// TwinCAT 3 PLC project MCAG_PLC_Project
// ProgramVersion: 3.1.0.8
// libraries:
//   Tc2_MC2, * (Beckhoff Automation GmbH)
//   Tc2_Standard, * (Beckhoff Automation GmbH)
//   Tc2_System, * (Beckhoff Automation GmbH)
//   Tc2_Utilities, * (Beckhoff Automation GmbH)
//   Tc3_Interfaces, * (Beckhoff Automation GmbH)
//   Tc3_Module, * (Beckhoff Automation GmbH)
// project tree:
//   DUTs/ DUT_AxisStatus_v0_01.TcDUT (not stored), DUT_AxisStatus_v0_02.TcDUT (not stored)
//   / PlcTask.TcTTO (not stored)
//   POUs/ FB_ReadFloatParameter.TcPOU (not stored), FB_ReadParameterInNc_v1_00.TcPOU (not stored), FB_WriteParameterInNc_v1_00.TcPOU (not stored), MAIN.TcPOU
//   POUs/Hardware/EtherCAT_Terminals/Analog_Inputs/ FB_CalculateFrequency_3702_v0_01.TcPOU (not stored), FB_EL3702_v0_00.TcPOU (not stored), FB_EL3773_v0_00.TcPOU (not stored), FB_EL3773_v1_00.TcPOU (not stored)
//   POUs/Hardware/EtherCAT_Terminals/Digital_Inputs/ EL1002_v1_00.TcPOU (not stored), EL1004_v1_00.TcPOU (not stored), EL1008_v1_00.TcPOU (not stored), EL1012_v1_00.TcPOU (not stored), EL1014_v1_00.TcPOU (not stored), EL1018_v1_00.TcPOU (not stored), EL1024_v1_00.TcPOU (not stored), EL1034_v1_00.TcPOU (not stored), EL1084_v1_00.TcPOU (not stored), EL1088_v1_00.TcPOU (not stored), EL1094_v1_00.TcPOU (not stored), EL1098_v1_00.TcPOU (not stored), EL1104_v1_00.TcPOU (not stored), EL1114_v1_00.TcPOU (not stored), EL1124_v1_00.TcPOU (not stored), EL1134_v1_00.TcPOU (not stored), EL1144_v1_00.TcPOU (not stored), EL1202_v1_00.TcPOU (not stored), EL1252_v1_00.TcPOU (not stored), EL1258_v0_00.TcPOU (not stored), EL1259_v0_00.TcPOU (not stored), EL1262_v0_00.TcPOU (not stored), EL1502_v0_00.TcPOU (not stored), EL1512_v0_00.TcPOU (not stored), EL1702_v1_00.TcPOU (not stored), EL1712_v1_00.TcPOU (not stored), EL1722_v1_00.TcPOU (not stored), EL1804_v1_00.TcPOU (not stored), EL1808_v1_00.TcPOU (not stored), EL1809_v1_00.TcPOU (not stored), EL1814_v1_00.TcPOU (not stored), EL1819_v1_00.TcPOU (not stored), EL1859_v1_00.TcPOU (not stored), EL1862_v1_00.TcPOU (not stored), EL1872_v1_00.TcPOU (not stored), EL1889_v1_00.TcPOU (not stored), FB_EL1008_v1_00.TcPOU (not stored), FB_EL1202_v1_00.TcPOU (not stored), FB_EL1252ASM_v1_00.TcPOU (not stored), FB_EL1252_v1_00.TcPOU (not stored)
//   POUs/Hardware/EtherCAT_Terminals/Digital_Outputs/ EL2002_v1_00.TcPOU (not stored), EL2004_v1_00.TcPOU (not stored), EL2008_v1_00.TcPOU (not stored), EL2022_v1_00.TcPOU (not stored), EL2024_v1_00.TcPOU (not stored), EL2032_v1_00.TcPOU (not stored), EL2034_v1_00.TcPOU (not stored), EL2042_v1_00.TcPOU (not stored), EL2084_v1_00.TcPOU (not stored), EL2088_v1_00.TcPOU (not stored), EL2124_v1_00.TcPOU (not stored), EL2202_v0_00.TcPOU (not stored), EL2212_v0_00.TcPOU (not stored), EL2252_v0_00.TcPOU (not stored), EL2258_v0_00.TcPOU (not stored), EL2262_v0_00.TcPOU (not stored), EL2502_v0_00.TcPOU (not stored), EL2521_v1_00.TcPOU (not stored), EL2535_v0_00.TcPOU (not stored), FB_EL2008_v1_00.TcPOU (not stored)
//   POUs/Hardware/EtherCAT_Terminals/Digital_Outputs/External_Types/ dutEL2521_Ctrl.TcDUT (not stored), dutEL2521_Status.TcDUT (not stored)
//   POUs/Hardware/EtherCAT_Terminals/Digital_Outputs/Safety_Terminals/ EL1904_v0_00.TcPOU (not stored), EL1908_v0_00.TcPOU (not stored), EL2901_v0_00.TcPOU (not stored), EL2902_v0_00.TcPOU (not stored), EL2904_v0_00.TcPOU (not stored), EL2964_v0_00.TcPOU (not stored), EL6900_v0_00.TcPOU (not stored), FB_EL1904_v1_00.TcPOU (not stored), FB_EL2904_v1_00.TcPOU (not stored), FB_EL6900_v1_00.TcPOU (not stored)
//   POUs/Hardware/EtherCAT_Terminals/Motion/ EL7211_v1_00.TcPOU (not stored), EL9576_v1_00.TcPOU (not stored)
//   POUs/Hardware/EtherCAT_Terminals/System/ EL9505_V1_00.TcPOU (not stored)
//   POUs/Hardware/Other/ EK1200.TcPOU (not stored)
//   POUs/Motion/ FB_DriveVirtual.TcPOU (not stored), FB_NcAxis.TcPOU (not stored)
// real-time tasks:
//   TASK PlcTask: cycle T#10ms, priority 20, ADS port 350
//   TASK PlcTaskCom: cycle T#1ms, priority 26, ADS port 351
// motion (NC):
//   TASK NC-Task 1 SAF: cycle T#2ms, priority 4, ADS port 501
//   TASK NC-Task 1 SVB: cycle T#10ms, priority 8, ADS port 511
//   AXIS Axis 1 (id 1)
//     Velo: RefSearch=10, RefSync=5
//     PositionAreaControl: Enable=false, RefSearch=false
//     OtherSettings: AllowMotionCmdToSlave=true
//     encoder EncType=8
//       EncPara: ScaleFactorNumerator=60, ScaleFactorDenominator=12800, MaxCount=#xffffffff
//     encoder EncId=129, EncType=4
//       EncPara: ScaleFactorNumerator=70, ScaleFactorDenominator=4096, Inverse=true, MaxCount=#x0000ffff
//         Inc: RefMode=2, RefSoftSyncMask=#x0000ffff
//     drive DrvType=9
//       DrvPara: MaxCount=#xffffffff, DriveControlDWord=#x00030100
//         Analog: VeloScale=1.02400649589962
//         TimeComp: TaskDelayCycles=1
//     controller CtrType=1
//       CtrPara: PriorControlFactor=1
//         PosDiffControl: Enable=false
//         PID: PosKp=10
//         Observer: BandWidth=20
//   AXIS Axis 2 (id 2)
//     OtherSettings: AllowMotionCmdToSlave=true
//     encoder EncType=8
//       EncPara: MaxCount=#x0036ee7f
//     drive DrvType=9
//       DrvPara: MaxCount=#xffffffff
//         Analog: VeloScale=6
//         TimeComp: TaskDelayCycles=1
//     controller CtrType=1
//       CtrPara: PriorControlFactor=1
//         Observer: BandWidth=20
//   AXIS Axis 3 (id 3)
//     OtherSettings: AllowMotionCmdToSlave=true
//     encoder EncType=1
//     drive DrvType=5
//       TimeComp: TaskDelayCycles=1
//     controller CtrType=1
//       CtrPara: PriorControlFactor=1
//         Observer: BandWidth=20
//   AXIS Axis 4 (id 4)
//     OtherSettings: AllowMotionCmdToSlave=true
//     encoder EncType=8
//       EncPara: MaxCount=#xffffffff
//     drive DrvType=9
//       DrvPara: MaxCount=#xffffffff, DriveControlDWord=#x00030100
//         Analog: VeloScale=1.02400649589962
//         TimeComp: TaskDelayCycles=1
//     controller CtrType=1
//       CtrPara: PriorControlFactor=1
//         Observer: BandWidth=20
// I/O:
//   DEVICE Device 1 (EtherCAT), AmsNetId 5.29.123.218.2.1
//     Term 1 (EK1200) [EK1200-5000 EtherCAT Power supply (2A E-Bus)]
//       Term 2 (EK1110) [EK1110 EtherCAT extension]
//     Drive 3 (AX5021-0000-0001) [AX5021-0000 EtherCAT Drive (SoE, 1 Ch.)]
//     Drive 4 (AX5112-0000-0203) [AX5112-0000-0203 EtherCAT Drive (SoE, 1 Ch.)]
//     Drive 5 (AX5112-0000-0203) [AX5112-0000-0203 EtherCAT Drive (SoE, 1 Ch.)]
// variable links:
//   NC-Task 1 SAF/Axes/Axis 1 <-> Device 1 (EtherCAT)/Drive 4 (AX5112-0000-0203)
//     Drive/Inputs/In/nDataIn1 <-> AT/Following distance
//     Drive/Inputs/In/nDcOutputTime <-> InfoData/DcOutputShift
//     Drive/Inputs/In/nState1 <-> AT/Drive status word @bit 8
//     Drive/Inputs/In/nState2 <-> AT/Drive status word
//     Drive/Inputs/In/nState4 @bit 1 <-> WcState/InputToggle
//     Drive/Inputs/In/nState4 <-> WcState/WcState
//     Drive/Outputs/Out/nCtrl1 <-> MDT/Master control word @bit 8
//     Drive/Outputs/Out/nDataOut1 <-> MDT/Position command value
//     Enc/Inputs/In/nDataIn1 <-> AT/Position feedback 1 value
//     Enc/Inputs/In/nDcInputTime <-> InfoData/DcInputShift
//     Enc/Inputs/In/nState4 @bit 1 <-> WcState/InputToggle
//     Enc/Inputs/In/nState4 <-> WcState/WcState
//   NC-Task 1 SAF/Axes/Axis 2 <-> Device 1 (EtherCAT)/Drive 3 (AX5021-0000-0001)
//     Drive/Inputs/In/nDcOutputTime <-> InfoData/DcOutputShift
//     Drive/Inputs/In/nState1 <-> AT/Drive status word @bit 8
//     Drive/Inputs/In/nState2 <-> AT/Drive status word
//     Drive/Inputs/In/nState4 @bit 1 <-> WcState/InputToggle
//     Drive/Inputs/In/nState4 <-> WcState/WcState
//     Drive/Outputs/Out/nCtrl1 <-> MDT/Master control word @bit 8
//     Enc/Inputs/In/nDcInputTime <-> InfoData/DcInputShift
//     Enc/Inputs/In/nState4 @bit 1 <-> WcState/InputToggle
//     Enc/Inputs/In/nState4 <-> WcState/WcState
//   NC-Task 1 SAF/Axes/Axis 4 <-> Device 1 (EtherCAT)/Drive 5 (AX5112-0000-0203)
//     Drive/Inputs/In/nDataIn1 <-> AT/Following distance
//     Drive/Inputs/In/nDcOutputTime <-> InfoData/DcOutputShift
//     Drive/Inputs/In/nState1 <-> AT/Drive status word @bit 8
//     Drive/Inputs/In/nState2 <-> AT/Drive status word
//     Drive/Inputs/In/nState4 @bit 1 <-> WcState/InputToggle
//     Drive/Inputs/In/nState4 <-> WcState/WcState
//     Drive/Outputs/Out/nCtrl1 <-> MDT/Master control word @bit 8
//     Drive/Outputs/Out/nDataOut1 <-> MDT/Position command value
//     Enc/Inputs/In/nDataIn1 <-> AT/Position feedback 1 value
//     Enc/Inputs/In/nDcInputTime <-> InfoData/DcInputShift
//     Enc/Inputs/In/nState4 @bit 1 <-> WcState/InputToggle
//     Enc/Inputs/In/nState4 <-> WcState/WcState
//   MCAG_PLC_Project/MCAG_PLC_Project Instance <-> NC-Task 1 SAF/Axes/Axis 1
//     PlcTask Inputs/MAIN.M1Link.Axis.NcToPlc <-> Outputs/ToPlc
//     PlcTask Outputs/MAIN.M1Link.Axis.PlcToNc <-> Inputs/FromPlc

// ---- POUs/MAIN.TcPOU
PROGRAM MAIN
VAR
	sVersion: STRING:='1.0.0';
	M1:FB_DriveVirtual;
	M1Link:FB_NcAxis;
	M2:FB_DriveVirtual;
	M2Link:FB_NcAxis;
	bLimitFwd AT %I*: BOOL;
	bLimitBwd AT %I*: BOOL;
	bHomeSensor AT %I*: BOOL;
END_VAR

act();

ACTION ACT:
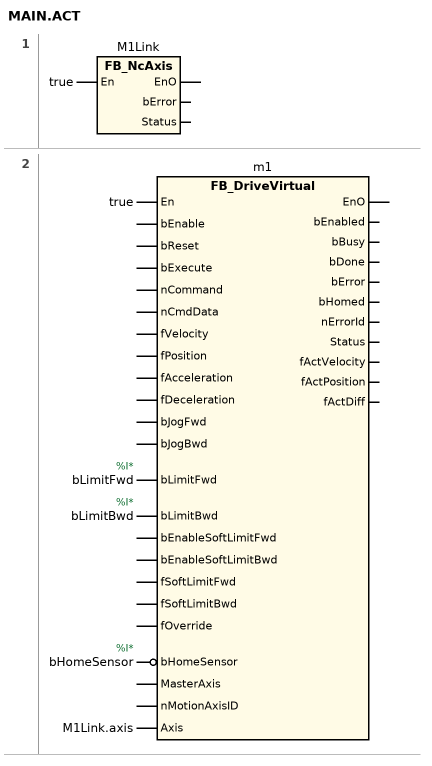
// NETWORK 1
M1Link(En := true); // FB_NcAxis

// NETWORK 2
//   bLimitFwd: AT %I*
//   bLimitBwd: AT %I*
//   bHomeSensor: AT %I*
m1(
    En := true,
    bLimitFwd := bLimitFwd,
    bLimitBwd := bLimitBwd,
    bHomeSensor := NOT bHomeSensor,
    Axis := M1Link.axis); // FB_DriveVirtual
END_ACTION

END_PROGRAM
